Yaskawa INFORM job: POSICAO_INICIAL_E_CAMERA.JBI

/JOB
//NAME MOV_IMG_H
//POS
///NPOS 2,0,0,0,0,0
///TOOL 1
///USER 10
///POSTYPE USER
///RECTAN
///RCONF 0,0,0,0,0,0,0,0
C00000=330.163,250.900,214.789,179.5565,0.1831,0.3047
C00001=244.171,268.622,582.664,179.5565,0.1831,0.3047
//INST
///DATE 2017/14/12 08:00
///ATTR SC,RW,RJ
///GROUP1 RB1
NOP
MOVL C00000 V=41.7
MOVL C00001 V=41.7
END
